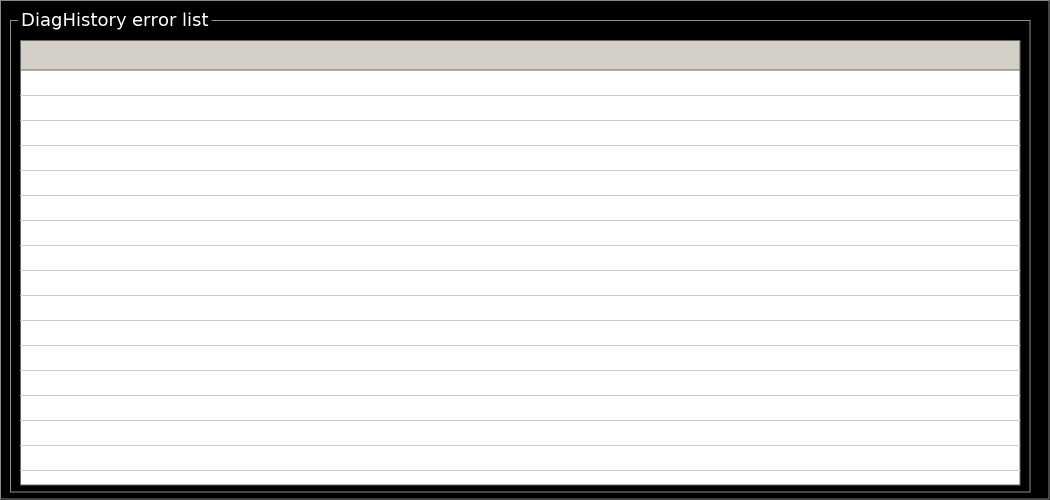
VISUALIZATION PH_SafeDiag_DiagHistory_black  // 1050x500
    GroupBox (10,12 1020x480), "DiagHistory error list"
        Table (10,28 1000x445), data array: P_Sample.stSafeDiag.arrDiagHistory
            p3854506369: P_Sample.stSafeDiag.arrDiagHistory[INDEX].EventID
            p1892666644: P_Sample.stSafeDiag.arrDiagHistory[INDEX].EventText
            p338671338: P_Sample.stSafeDiag.arrDiagHistory[INDEX].Severity
            p2170511999: P_Sample.stSafeDiag.arrDiagHistory[INDEX].TimeRaised
            p3723444502: MAINSafety.stEL6910.stVisu
END_VISUALIZATION

(* stored: Version 1.1.0.1, ProductVersion 3.1.4024.12
   Visu PH_SafeDiag_DiagHistory_black: Id {601f83b5-da4b-45db-ac64-2bb4c263afaa} *)
